KUKA KRL program: chk_w6_grp3_opn.src

&ACCESS RV4
&COMMENT Check GRP AXOR Z3 OPEN
DEF chk_w6_grp3_opn( )

; Check gripper axor OPEN Z3.1
;//---- Start User-------

$TIMER[10] = 0
$TIMER_STOP[10] = FALSE

WAIT FOR ($IN[497])
WAIT FOR (NOT $IN[498])

$TIMER_STOP[10] = TRUE
$TIMER[10] = 0

;//---- End User---------
END
